(* Logix 5000 project; controller Kollmeyer_LiveDemo_TBENLX8IOL_TBIL vendor 1 type 14 code 176 rev 32.11; software revision 32.00; part 9 of 9 *)
(* tags used below, declared in another part *)
   CommonData : Turck_IOL_CommonData;
   Port1_VID : DINT;
   Port1_DID : DINT;
   Port2_VID : DINT;
   Port2_DID : DINT;
   Port3_VID : DINT;
   Port3_DID : DINT;
   Port4_VID : DINT;
   Port4_DID : DINT;
   Port5_VID : DINT;
   Port5_DID : DINT;
   Port6_VID : DINT;
   Port6_DID : DINT;
   Port7_VID : DINT;
   Port7_DID : DINT;
   Port8_VID : DINT;
   Port8_DID : DINT;
   IOLS1 : BOOL;
   IOLS2 : BOOL;
   IOLS3 : BOOL;
   IOLS4 : BOOL;
   IOLS5 : BOOL;
   IOLS6 : BOOL;
   IOLS7 : BOOL;
   IOLReadActive : BOOL;
   IOLWriteActive : BOOL;
   Retry : BOOL;
   RetryCount : DINT;
   IOLS4_Bad : BOOL;
   IOL_S2_0_Count : DINT;
   IOL_S6_0_Count : DINT;
   Busy_Retry : BOOL;
   IOL_S2_0_Total : DINT;
   IOL_S3_Retry : DINT;
   IOL_S1_Count : DINT;
   IOL_S2_Count : DINT;
   IOL_S3_Count : DINT;
   IOL_S5_Count : DINT;
   IOL_S6_Count : DINT;
   IOL_S6_NotBusy_Count : DINT;
   RetryTotal : DINT;
   IOL_S4_Bad_Count : DINT;
   IOL_S2_Error_Count : DINT;
   IOL_Done_Count : DINT;
   IOL_Error_Count : DINT;
   IOLReset_ONS : BOOL;
   IOLS2A : BOOL;
   IOLS5A : BOOL;
   Busy_Response : BOOL;
   READ_PORT_DATA : IOL_ReadString;
(* TBEN_L_8IOL_AOI, continued *)

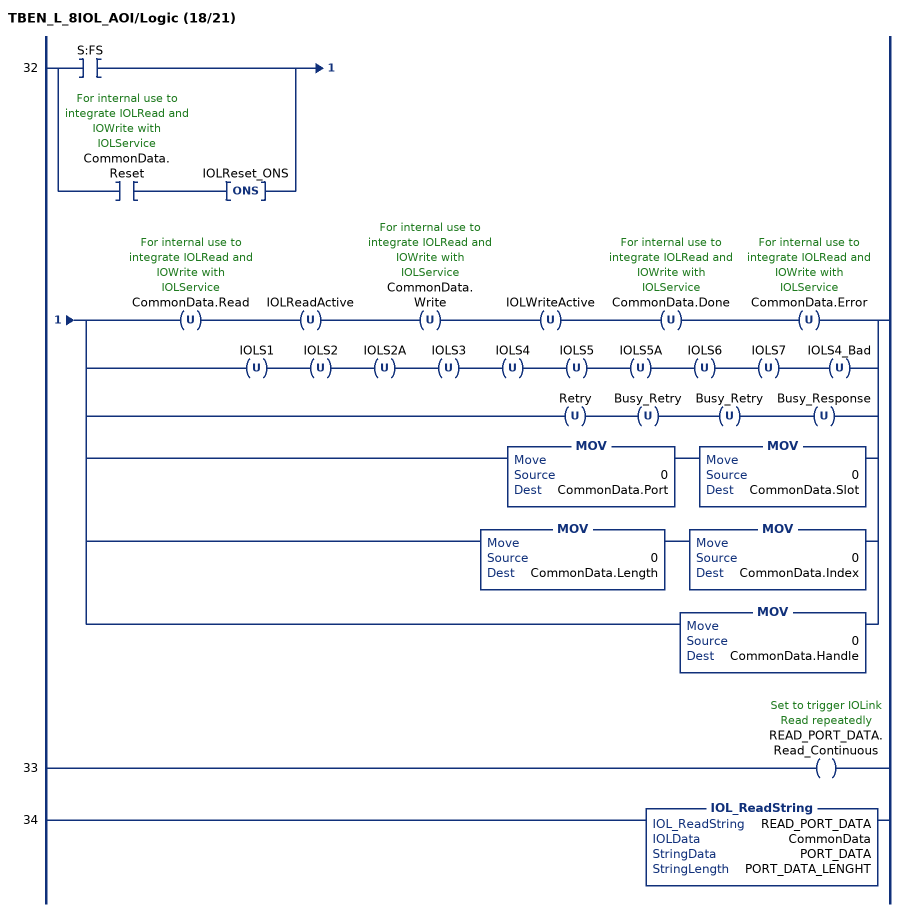
   32: [XIC(S:FS) ,XIC(CommonData.Reset) ONS(IOLReset_ONS) ][OTU(CommonData.Read) OTU(IOLReadActive) OTU(CommonData.Write) OTU(IOLWriteActive) OTU(CommonData.Done) OTU(CommonData.Error) ,OTU(IOLS1) OTU(IOLS2) OTU(IOLS2A) OTU(IOLS3) OTU(IOLS4) OTU(IOLS5) OTU(IOLS5A) OTU(IOLS6) OTU(IOLS7) OTU(IOLS4_Bad) ,OTU(Retry) OTU(Busy_Retry) OTU(Busy_Retry) OTU(Busy_Response) ,MOV(0,CommonData.Port) MOV(0,CommonData.Slot) ,MOV(0,CommonData.Length) MOV(0,CommonData.Index) ,MOV(0,CommonData.Handle) ];
   33: OTE(READ_PORT_DATA.Read_Continuous);
   34: IOL_ReadString(READ_PORT_DATA,CommonData,PORT_DATA,PORT_DATA_LENGHT);
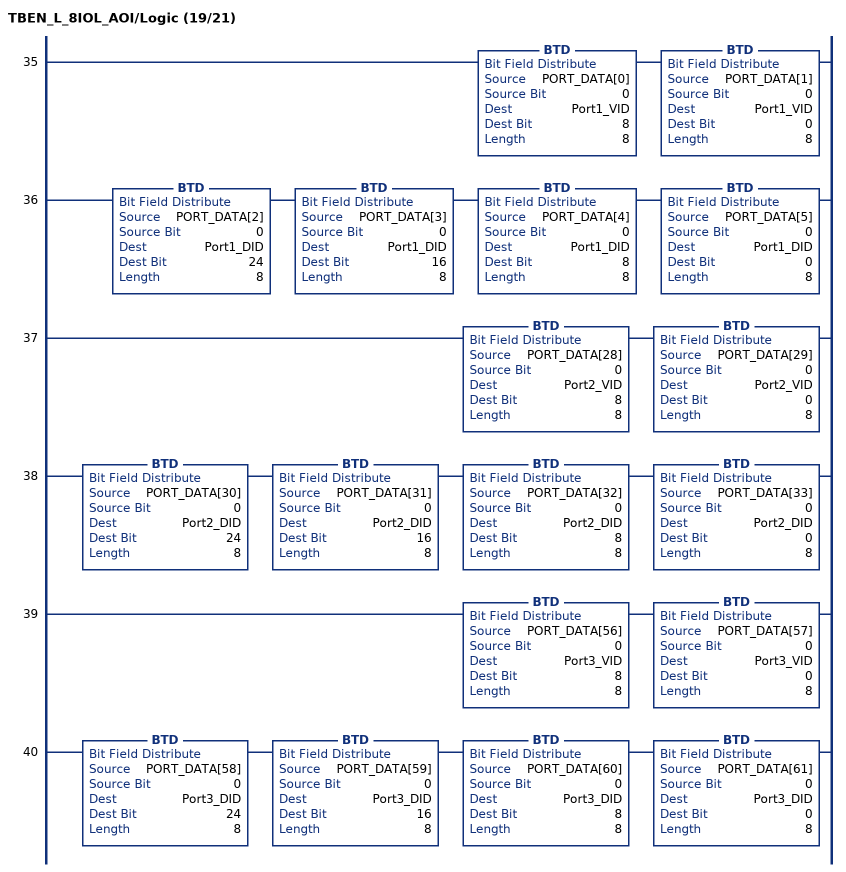
   35: BTD(PORT_DATA[0],0,Port1_VID,8,8)BTD(PORT_DATA[1],0,Port1_VID,0,8);
   36: BTD(PORT_DATA[2],0,Port1_DID,24,8)BTD(PORT_DATA[3],0,Port1_DID,16,8)BTD(PORT_DATA[4],0,Port1_DID,8,8)BTD(PORT_DATA[5],0,Port1_DID,0,8);
   37: BTD(PORT_DATA[28],0,Port2_VID,8,8)BTD(PORT_DATA[29],0,Port2_VID,0,8);
   38: BTD(PORT_DATA[30],0,Port2_DID,24,8)BTD(PORT_DATA[31],0,Port2_DID,16,8)BTD(PORT_DATA[32],0,Port2_DID,8,8)BTD(PORT_DATA[33],0,Port2_DID,0,8);
   39: BTD(PORT_DATA[56],0,Port3_VID,8,8)BTD(PORT_DATA[57],0,Port3_VID,0,8);
   40: BTD(PORT_DATA[58],0,Port3_DID,24,8)BTD(PORT_DATA[59],0,Port3_DID,16,8)BTD(PORT_DATA[60],0,Port3_DID,8,8)BTD(PORT_DATA[61],0,Port3_DID,0,8);
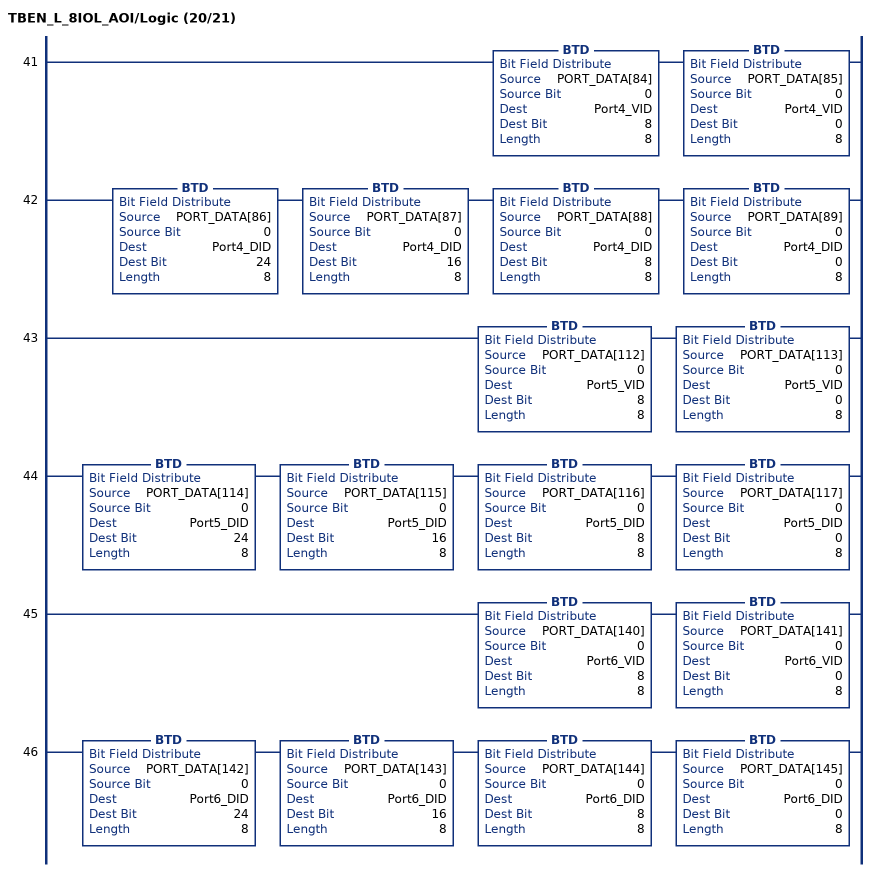
   41: BTD(PORT_DATA[84],0,Port4_VID,8,8)BTD(PORT_DATA[85],0,Port4_VID,0,8);
   42: BTD(PORT_DATA[86],0,Port4_DID,24,8)BTD(PORT_DATA[87],0,Port4_DID,16,8)BTD(PORT_DATA[88],0,Port4_DID,8,8)BTD(PORT_DATA[89],0,Port4_DID,0,8);
   43: BTD(PORT_DATA[112],0,Port5_VID,8,8)BTD(PORT_DATA[113],0,Port5_VID,0,8);
   44: BTD(PORT_DATA[114],0,Port5_DID,24,8)BTD(PORT_DATA[115],0,Port5_DID,16,8)BTD(PORT_DATA[116],0,Port5_DID,8,8)BTD(PORT_DATA[117],0,Port5_DID,0,8);
   45: BTD(PORT_DATA[140],0,Port6_VID,8,8)BTD(PORT_DATA[141],0,Port6_VID,0,8);
   46: BTD(PORT_DATA[142],0,Port6_DID,24,8)BTD(PORT_DATA[143],0,Port6_DID,16,8)BTD(PORT_DATA[144],0,Port6_DID,8,8)BTD(PORT_DATA[145],0,Port6_DID,0,8);
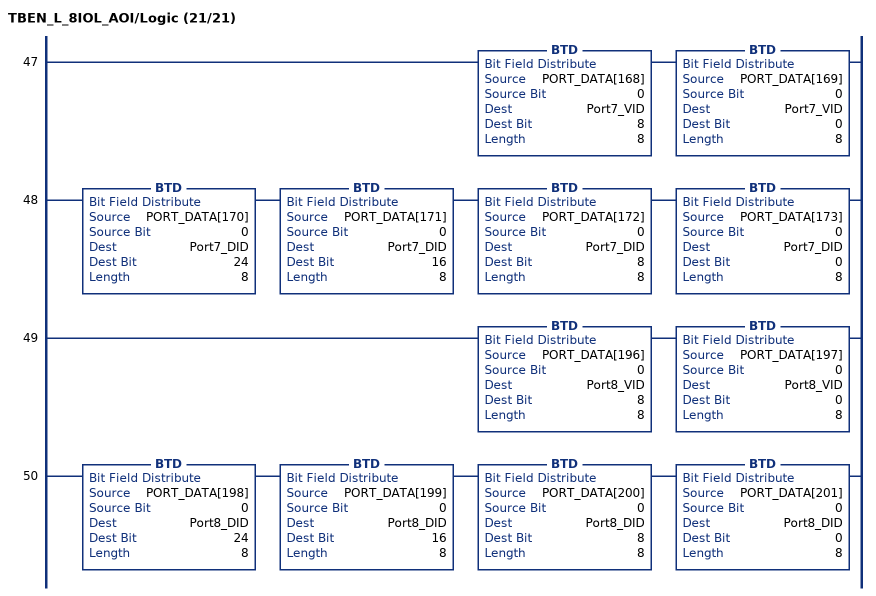
   47: BTD(PORT_DATA[168],0,Port7_VID,8,8)BTD(PORT_DATA[169],0,Port7_VID,0,8);
   48: BTD(PORT_DATA[170],0,Port7_DID,24,8)BTD(PORT_DATA[171],0,Port7_DID,16,8)BTD(PORT_DATA[172],0,Port7_DID,8,8)BTD(PORT_DATA[173],0,Port7_DID,0,8);
   49: BTD(PORT_DATA[196],0,Port8_VID,8,8)BTD(PORT_DATA[197],0,Port8_VID,0,8);
   50: BTD(PORT_DATA[198],0,Port8_DID,24,8)BTD(PORT_DATA[199],0,Port8_DID,16,8)BTD(PORT_DATA[200],0,Port8_DID,8,8)BTD(PORT_DATA[201],0,Port8_DID,0,8);
END_ROUTINE

ROUTINE Prescan   (* ladder *)
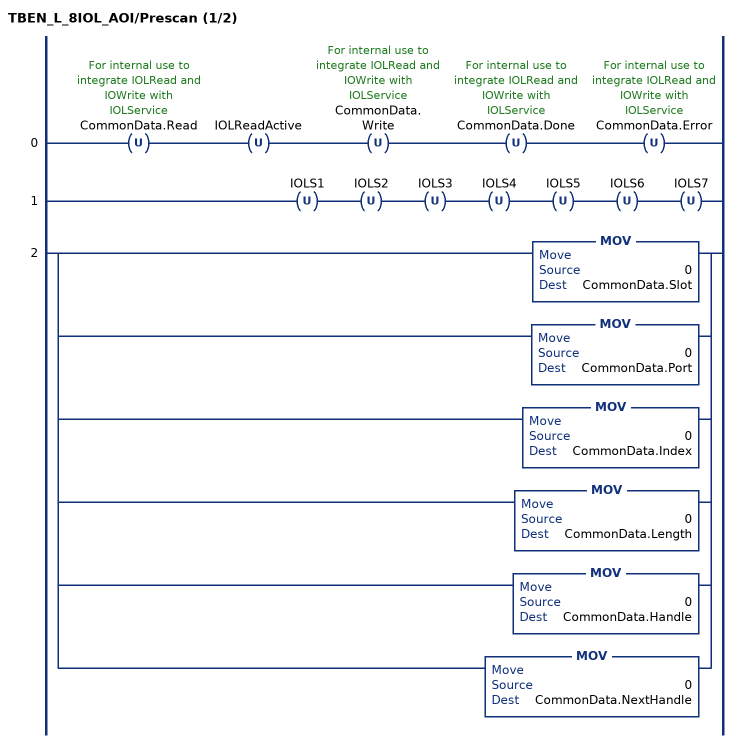
   0: OTU(CommonData.Read)OTU(IOLReadActive)OTU(CommonData.Write)OTU(CommonData.Done)OTU(CommonData.Error);
   1: OTU(IOLS1)OTU(IOLS2)OTU(IOLS3)OTU(IOLS4)OTU(IOLS5)OTU(IOLS6)OTU(IOLS7);
   2: [MOV(0,CommonData.Slot) ,MOV(0,CommonData.Port) ,MOV(0,CommonData.Index) ,MOV(0,CommonData.Length) ,MOV(0,CommonData.Handle) ,MOV(0,CommonData.NextHandle) ];
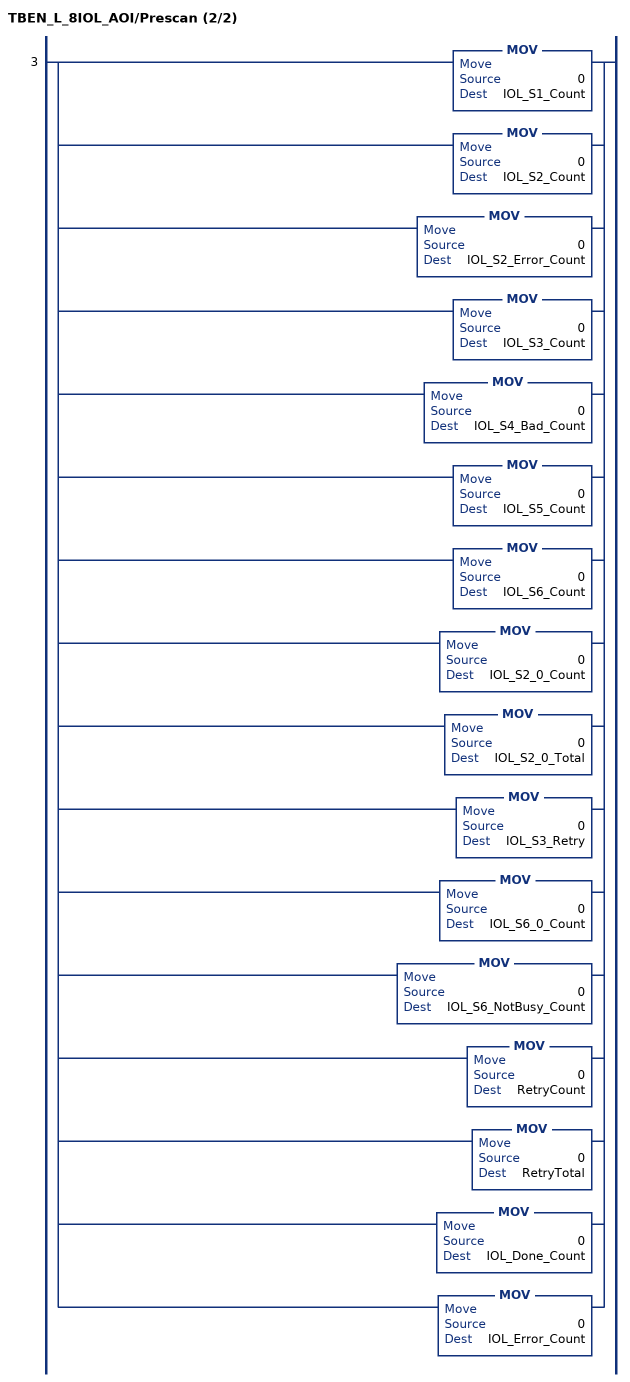
   3: [MOV(0,IOL_S1_Count) ,MOV(0,IOL_S2_Count) ,MOV(0,IOL_S2_Error_Count) ,MOV(0,IOL_S3_Count) ,MOV(0,IOL_S4_Bad_Count) ,MOV(0,IOL_S5_Count) ,MOV(0,IOL_S6_Count) ,MOV(0,IOL_S2_0_Count) ,MOV(0,IOL_S2_0_Total) ,MOV(0,IOL_S3_Retry) ,MOV(0,IOL_S6_0_Count) ,MOV(0,IOL_S6_NotBusy_Count) ,MOV(0,RetryCount) ,MOV(0,RetryTotal) ,MOV(0,IOL_Done_Count) ,MOV(0,IOL_Error_Count) ];
END_ROUTINE
END_ADD_ON_INSTRUCTION

ADD_ON_INSTRUCTION TBIL_M1_16DXP_Pro   (* revision 1.0 *)
// TBIL-M1-16DXP AOI with Acyclic Index Data
VAR_INPUT
   Port : INT; {visible}
END_VAR
VAR_OUTPUT
   IN1A : BOOL; {access Read Only, visible}
   IN1B : BOOL; {visible}
   IN2A : BOOL; {visible}
   IN2B : BOOL; {visible}
   IN3A : BOOL; {visible}
   IN3B : BOOL; {visible}
   IN4A : BOOL; {visible}
   IN4B : BOOL; {visible}
   IN5A : BOOL; {visible}
   IN5B : BOOL; {visible}
   IN6A : BOOL; {visible}
   IN6B : BOOL; {visible}
   IN7A : BOOL; {visible}
   IN7B : BOOL; {visible}
   IN8A : BOOL; {visible}
   IN8B : BOOL; {visible}
END_VAR
VAR_INPUT
   OUT1A : BOOL; {visible}
   OUT1B : BOOL; {visible}
   OUT2A : BOOL; {visible}
   OUT2B : BOOL; {visible}
   OUT3A : BOOL; {visible}
   OUT3B : BOOL; {visible}
   OUT4A : BOOL; {visible}
   OUT4B : BOOL; {visible}
   OUT5A : BOOL; {visible}
   OUT5B : BOOL; {visible}
   OUT6A : BOOL; {visible}
   OUT6B : BOOL; {visible}
   OUT7A : BOOL; {visible}
   OUT7B : BOOL; {visible}
   OUT8A : BOOL; {visible}
   OUT8B : BOOL; {visible}
END_VAR
VAR_OUTPUT
   V_ID : DINT;
   D_ID : DINT;
END_VAR
VAR_IN_OUT
   APPL_TAG : SINT[82]; {required}
   COMMON_DATA : Turck_IOL_CommonData; {required}
END_VAR
VAR_OUTPUT
   Wrong_Or_Missing_Device : BOOL; {access Read Only, visible}
END_VAR
VAR
   READ_APPL_TAG : IOL_ReadString := (Slot := 1, Port := 1, Index := 24); {access None}
   APPL_TAG_LENGHT : DINT; {access None}
   READ_DATA : IOL_ReadString := (Slot := 1, Port := 1); {access None}
   PORT_DATA : SINT[82]; {access None}
   PORT_DATA_LENGHT : DINT; {access None}
   READ_PROCESS_DATA : IOL_ReadString := (Slot := 1, Port := 1, Index := 40); {access None}
   PROCESS_DATA : SINT[82]; {access None}
   PROCESS_DATA_LENGHT : DINT; {access None}
   RAW_PROCESS_DATA : SINT[82]; {access None}
END_VAR

ROUTINE Logic   (* ladder *)
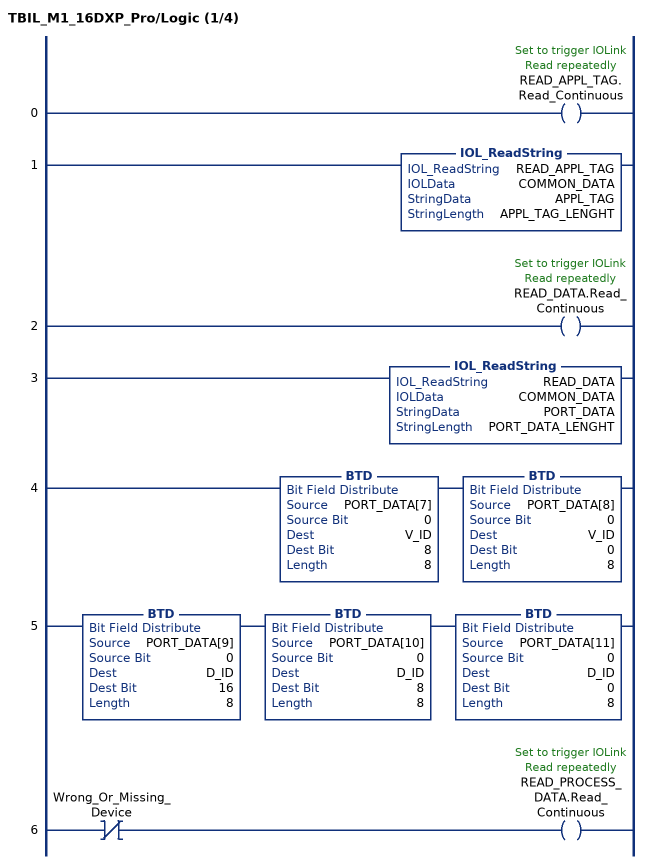
   0: OTE(READ_APPL_TAG.Read_Continuous);
   1: IOL_ReadString(READ_APPL_TAG,COMMON_DATA,APPL_TAG,APPL_TAG_LENGHT);
   2: OTE(READ_DATA.Read_Continuous);
   3: IOL_ReadString(READ_DATA,COMMON_DATA,PORT_DATA,PORT_DATA_LENGHT);
   4: BTD(PORT_DATA[7],0,V_ID,8,8)BTD(PORT_DATA[8],0,V_ID,0,8);
   5: BTD(PORT_DATA[9],0,D_ID,16,8)BTD(PORT_DATA[10],0,D_ID,8,8)BTD(PORT_DATA[11],0,D_ID,0,8);
   6: XIO(Wrong_Or_Missing_Device)OTE(READ_PROCESS_DATA.Read_Continuous);
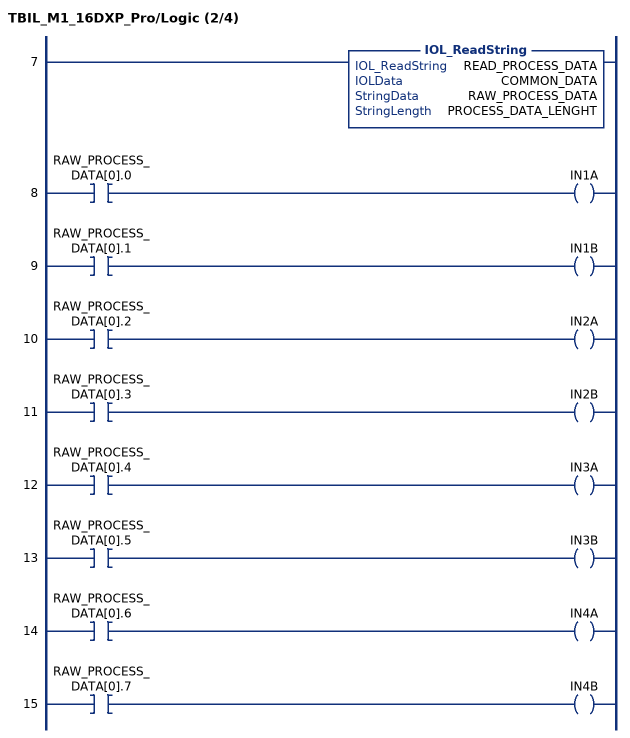
   7: IOL_ReadString(READ_PROCESS_DATA,COMMON_DATA,RAW_PROCESS_DATA,PROCESS_DATA_LENGHT);
   8: XIC(RAW_PROCESS_DATA[0].0)OTE(IN1A);
   9: XIC(RAW_PROCESS_DATA[0].1)OTE(IN1B);
   10: XIC(RAW_PROCESS_DATA[0].2)OTE(IN2A);
   11: XIC(RAW_PROCESS_DATA[0].3)OTE(IN2B);
   12: XIC(RAW_PROCESS_DATA[0].4)OTE(IN3A);
   13: XIC(RAW_PROCESS_DATA[0].5)OTE(IN3B);
   14: XIC(RAW_PROCESS_DATA[0].6)OTE(IN4A);
   15: XIC(RAW_PROCESS_DATA[0].7)OTE(IN4B);
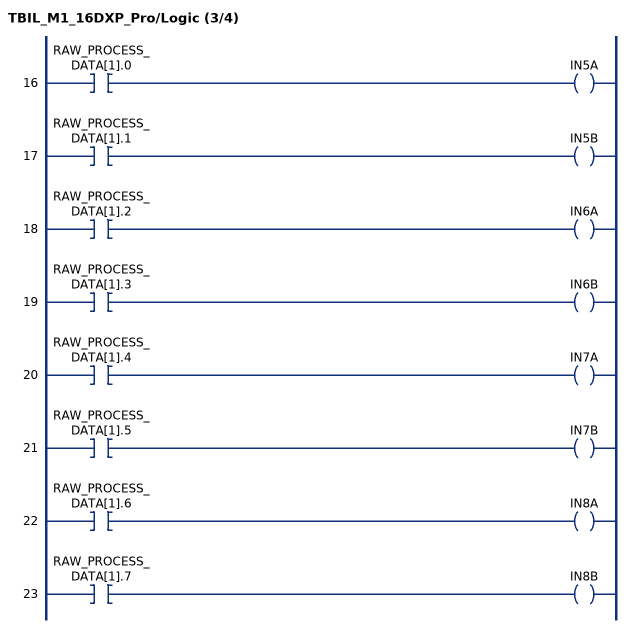
   16: XIC(RAW_PROCESS_DATA[1].0)OTE(IN5A);
   17: XIC(RAW_PROCESS_DATA[1].1)OTE(IN5B);
   18: XIC(RAW_PROCESS_DATA[1].2)OTE(IN6A);
   19: XIC(RAW_PROCESS_DATA[1].3)OTE(IN6B);
   20: XIC(RAW_PROCESS_DATA[1].4)OTE(IN7A);
   21: XIC(RAW_PROCESS_DATA[1].5)OTE(IN7B);
   22: XIC(RAW_PROCESS_DATA[1].6)OTE(IN8A);
   23: XIC(RAW_PROCESS_DATA[1].7)OTE(IN8B);
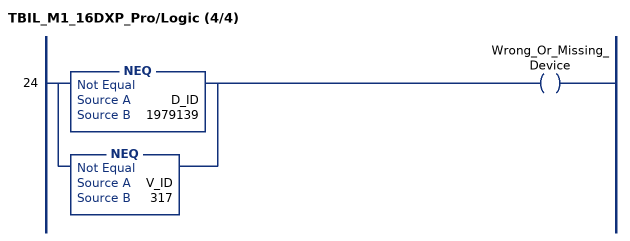
   24: [NEQ(D_ID,1979139) ,NEQ(V_ID,317) ]OTE(Wrong_Or_Missing_Device);
END_ROUTINE
END_ADD_ON_INSTRUCTION

ADD_ON_INSTRUCTION Turck_TBIL_16DXP   (* revision 1.0 *)
VAR_INPUT
   Process_Data_In : INT; {required}
END_VAR
VAR_OUTPUT
   Process_Data_Out : INT; {required}
   Input_1A : BOOL; {visible}
   Input_1B : BOOL; {visible}
   Input_2A : BOOL; {visible}
   Input_2B : BOOL; {visible}
   Input_3A : BOOL; {visible}
   Input_3B : BOOL; {visible}
   Input_4A : BOOL; {visible}
   Input_4B : BOOL; {visible}
   Input_5A : BOOL; {visible}
   Input_5B : BOOL; {visible}
   Input_6A : BOOL; {visible}
   Input_6B : BOOL; {visible}
   Input_7A : BOOL; {visible}
   Input_7B : BOOL; {visible}
   Input_8A : BOOL; {visible}
   Input_8B : BOOL; {visible}
END_VAR
VAR_INPUT
   Output_1A : BOOL; {visible}
   Output_1B : BOOL; {visible}
   Output_2A : BOOL; {visible}
   Output_2B : BOOL; {visible}
   Output_3A : BOOL; {visible}
   Output_3B : BOOL; {visible}
   Output_4A : BOOL; {visible}
   Output_4B : BOOL; {visible}
   Output_5A : BOOL; {visible}
   Output_5B : BOOL; {visible}
   Output_6A : BOOL; {visible}
   Output_6B : BOOL; {visible}
   Output_7A : BOOL; {visible}
   Output_7B : BOOL; {visible}
   Output_8A : BOOL; {visible}
   Output_8B : BOOL; {visible}
END_VAR

ROUTINE Logic   (* ladder *)
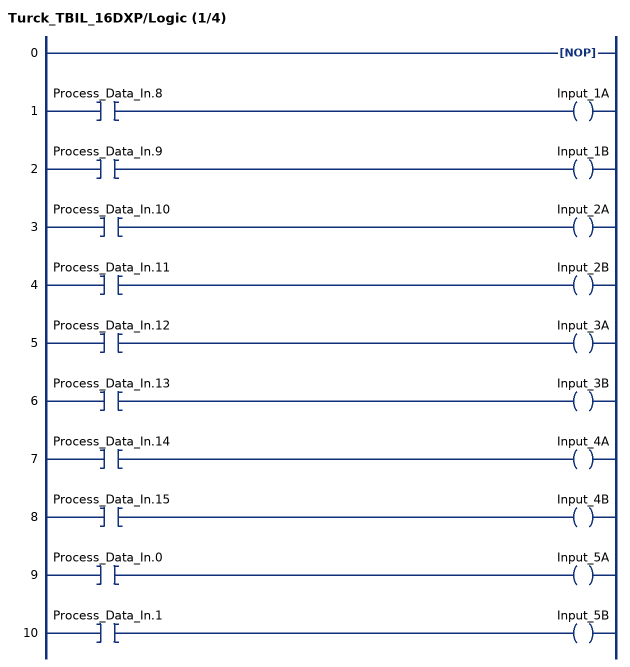
   0: NOP();
   1: XIC(Process_Data_In.8)OTE(Input_1A);
   2: XIC(Process_Data_In.9)OTE(Input_1B);
   3: XIC(Process_Data_In.10)OTE(Input_2A);
   4: XIC(Process_Data_In.11)OTE(Input_2B);
   5: XIC(Process_Data_In.12)OTE(Input_3A);
   6: XIC(Process_Data_In.13)OTE(Input_3B);
   7: XIC(Process_Data_In.14)OTE(Input_4A);
   8: XIC(Process_Data_In.15)OTE(Input_4B);
   9: XIC(Process_Data_In.0)OTE(Input_5A);
   10: XIC(Process_Data_In.1)OTE(Input_5B);
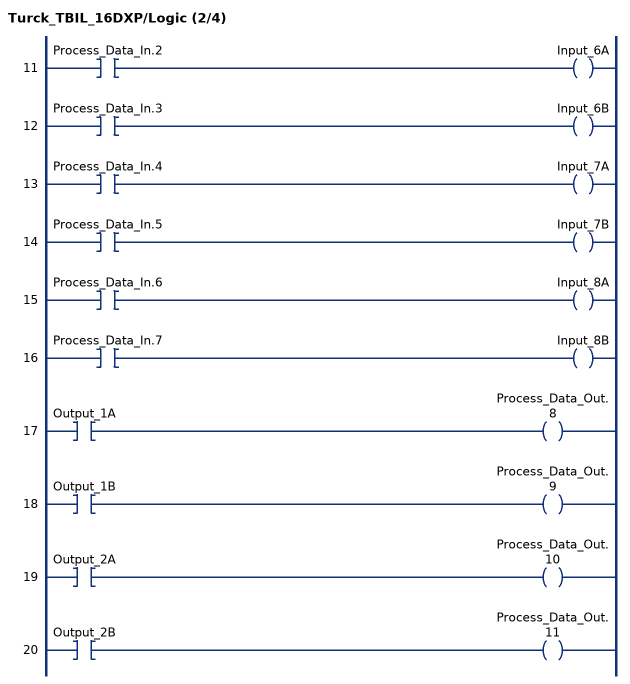
   11: XIC(Process_Data_In.2)OTE(Input_6A);
   12: XIC(Process_Data_In.3)OTE(Input_6B);
   13: XIC(Process_Data_In.4)OTE(Input_7A);
   14: XIC(Process_Data_In.5)OTE(Input_7B);
   15: XIC(Process_Data_In.6)OTE(Input_8A);
   16: XIC(Process_Data_In.7)OTE(Input_8B);
   17: XIC(Output_1A)OTE(Process_Data_Out.8);
   18: XIC(Output_1B)OTE(Process_Data_Out.9);
   19: XIC(Output_2A)OTE(Process_Data_Out.10);
   20: XIC(Output_2B)OTE(Process_Data_Out.11);
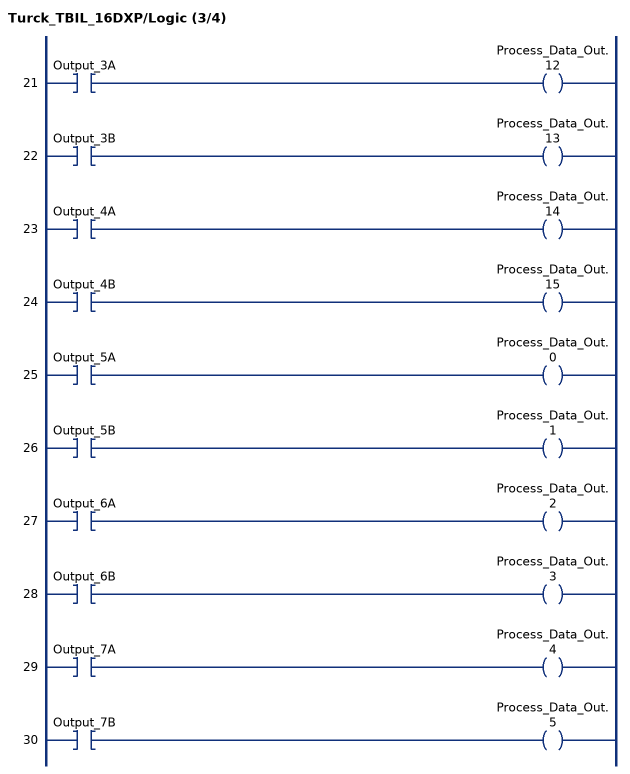
   21: XIC(Output_3A)OTE(Process_Data_Out.12);
   22: XIC(Output_3B)OTE(Process_Data_Out.13);
   23: XIC(Output_4A)OTE(Process_Data_Out.14);
   24: XIC(Output_4B)OTE(Process_Data_Out.15);
   25: XIC(Output_5A)OTE(Process_Data_Out.0);
   26: XIC(Output_5B)OTE(Process_Data_Out.1);
   27: XIC(Output_6A)OTE(Process_Data_Out.2);
   28: XIC(Output_6B)OTE(Process_Data_Out.3);
   29: XIC(Output_7A)OTE(Process_Data_Out.4);
   30: XIC(Output_7B)OTE(Process_Data_Out.5);
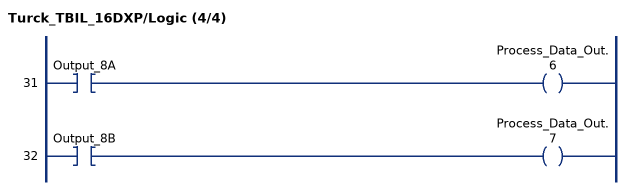
   31: XIC(Output_8A)OTE(Process_Data_Out.6);
   32: XIC(Output_8B)OTE(Process_Data_Out.7);
END_ROUTINE
END_ADD_ON_INSTRUCTION

VAR_GLOBAL   (* controller tags *)
   APPL_TAG_TBIL_PORT1 : SINT[82] := ([0] := 72, [1] := 69, [2] := 76, [3] := 76, [4] := 79, [5] := 32, [6] := 87, [7] := 79, [8] := 82, [9] := 76, [10] := 68);
   ENABLE_AOI : BOOL := 1;
   IOL_ReceiveMSG : MESSAGE;
        MessageParameters(ServiceCode := 16#000e, DestinationTag := TBEN_192_168_1_7_DATA.ReceiveData, ...)
   IOL_SendMSG : MESSAGE;
        MessageParameters(ServiceCode := 16#0010, LocalElement := TBEN_192_168_1_7_DATA.SendData, ...)
   TBEN_192_168_1_7 : TBEN_L_8IOL_AOI;
   TBEN_192_168_1_7_DATA : Turck_IOL_CommonData := (Read := 1, Slot := 1, Index := -1, SubIndex := 68, Length := 224, Status := 1016, NextHandle := 4, ReceiveData[0] := -3, ReceiveData[1] := 17, ReceiveData[2] := 8, ReceiveData[3] := 1, ReceiveData[4] := -2, ReceiveData[5] := 74, ReceiveData[6] := -128, ReceiveData[8] := 40, ReceiveData[12] := 16, SendData[1] := -4, SendData[2] := 17, SendData[3] := 8, SendData[5] := -2, SendData[6] := 74, SendData[7] := 3, SendData[8] := -1, SendData[9] := -1, SendData[10] := 68);
   TBEN_8IOL_1_Process_Data_In : Generic_173_Words;
   TBEN_8IOL_1_Process_Data_Out : Generic_131_Words;
   TBIL_PORT1 : TBIL_M1_16DXP_Pro := (Port := 1, IN3B := 1, V_ID := 16#0000_013d, D_ID := 16#001e_3303);
END_VAR

PROGRAM MainProgram   (* main routine MainRoutine *)

ROUTINE MainRoutine   (* ladder *)
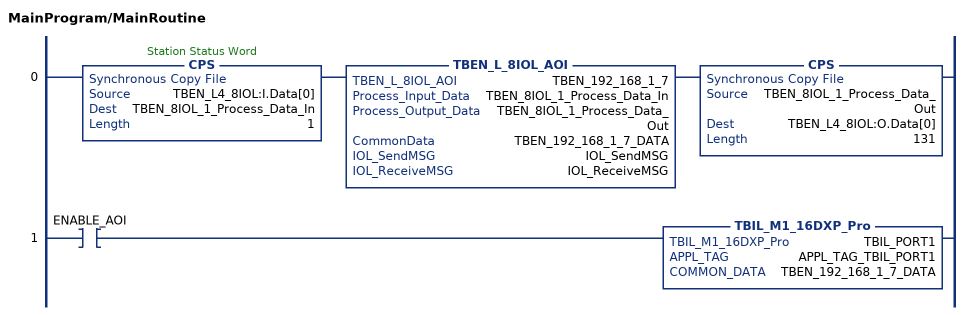
   0: CPS(TBEN_L4_8IOL:I.Data[0],TBEN_8IOL_1_Process_Data_In,1)TBEN_L_8IOL_AOI(TBEN_192_168_1_7,TBEN_8IOL_1_Process_Data_In,TBEN_8IOL_1_Process_Data_Out,TBEN_192_168_1_7_DATA,IOL_SendMSG,IOL_ReceiveMSG)CPS(TBEN_8IOL_1_Process_Data_Out,TBEN_L4_8IOL:O.Data[0],131);
   1: XIC(ENABLE_AOI)TBIL_M1_16DXP_Pro(TBIL_PORT1,APPL_TAG_TBIL_PORT1,TBEN_192_168_1_7_DATA);
END_ROUTINE
END_PROGRAM

PROGRAM SafetyProgram   (* main routine MainRoutine, safety *)

ROUTINE MainRoutine   (* ladder *)
END_ROUTINE
END_PROGRAM
